(* Logix 5000 project; controller cal1632 1756-L62 rev 16.20; software revision 16.05; part 41 of 61 *)
(* tags used below, declared in another part *)
   FAULT : BOOL;
   p01r09_pb_global_reset : BOOL;
   p02_dint_to_hmi : hmi_dint;
   p24_di_edge_guide_auto : BOOL;
   p24_di_edge_guide_center : BOOL;
   p24_di_edge_guide_left : BOOL;
   p24_di_edge_guide_right : BOOL;
   p24_dint_to_hmi : DINT[16];
   p24_do_edge_guide_input_1 : BOOL;
   p24r01 : routine;
   p24r02 : routine;
   p24r02_fault_exists : BOOL;
   p24r02_timer_fault : TIMER[4];
   p24r02_timer_warning : TIMER[4];
   p24r02_unack_fault : BOOL;
   p24r02_unack_warning : BOOL;
   p24r02_warning_exists : BOOL;
   p24r03 : routine;
   p24r03_timer_fault : TIMER[4];
   p24r03_timer_warning : TIMER[4];
   p24r04 : routine;
   p24r04_timer_fault : TIMER[4];
   p24r04_timer_warning : TIMER[4];
   p24r05 : routine;
   p24r05_timer_fault : TIMER[4];
   p24r05_timer_warning : TIMER[4];
   p24r06 : routine;
   p24r06_timer_fault : TIMER[4];
   p24r06_timer_warning : TIMER[4];
   p24r07 : routine;
   p24r07_timer_fault : TIMER[4];
   p24r07_timer_warning : TIMER[4];
   p24r08 : routine;
   p24r09 : routine;
   p24r10 : routine;

PROGRAM P24_Edge_Control   (* main routine R01_Main *)

ROUTINE R01_Main   (* ladder *)
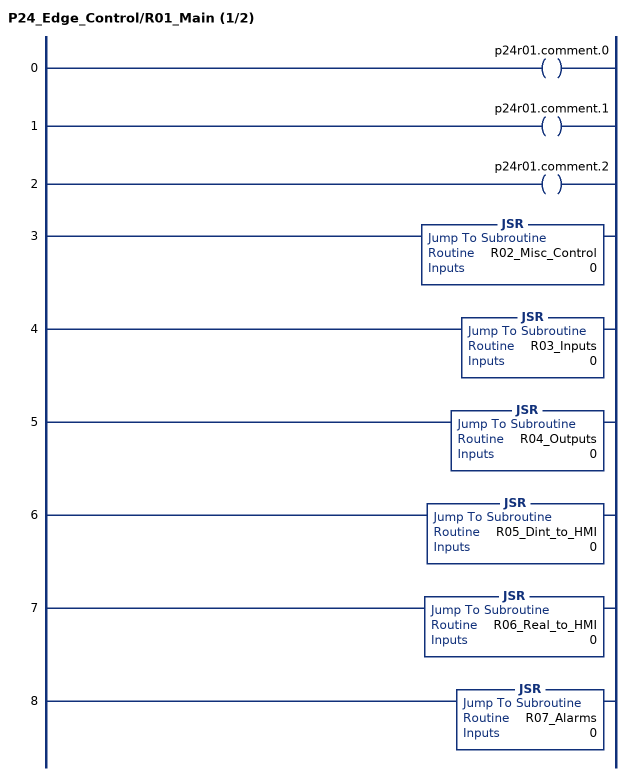
   0: OTE(p24r01.comment.0);
   1: OTE(p24r01.comment.1);
   2: OTE(p24r01.comment.2);
   3: JSR(R02_Misc_Control,0);
   4: JSR(R03_Inputs,0);
   5: JSR(R04_Outputs,0);
   6: JSR(R05_Dint_to_HMI,0);
   7: JSR(R06_Real_to_HMI,0);
   8: JSR(R07_Alarms,0);
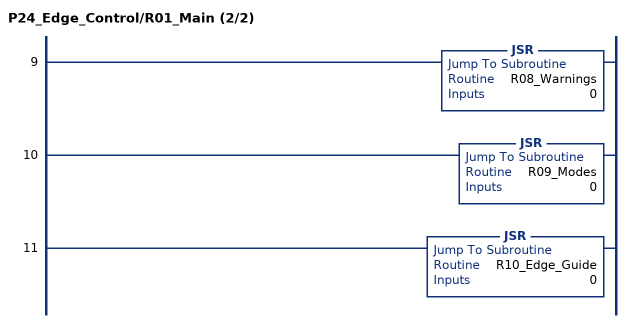
   9: JSR(R08_Warnings,0);
   10: JSR(R09_Modes,0);
   11: JSR(R10_Edge_Guide,0);
END_ROUTINE

ROUTINE R02_Misc_Control   (* ladder *)
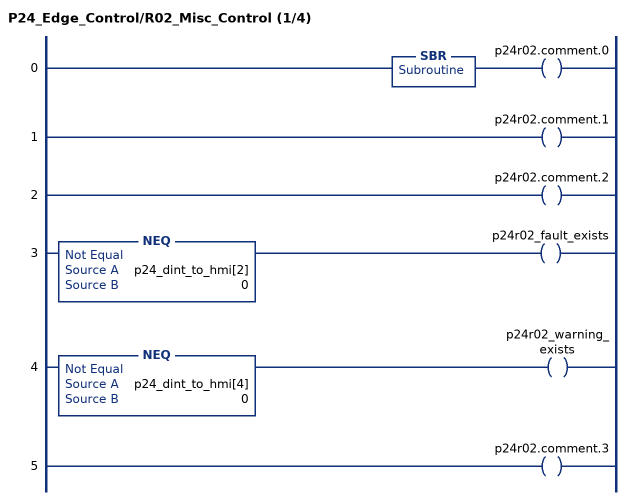
   0: SBR()OTE(p24r02.comment.0);
   1: OTE(p24r02.comment.1);
   2: OTE(p24r02.comment.2);
   3: NEQ(p24_dint_to_hmi[2],0)OTE(p24r02_fault_exists);
   4: NEQ(p24_dint_to_hmi[4],0)OTE(p24r02_warning_exists);
   5: OTE(p24r02.comment.3);
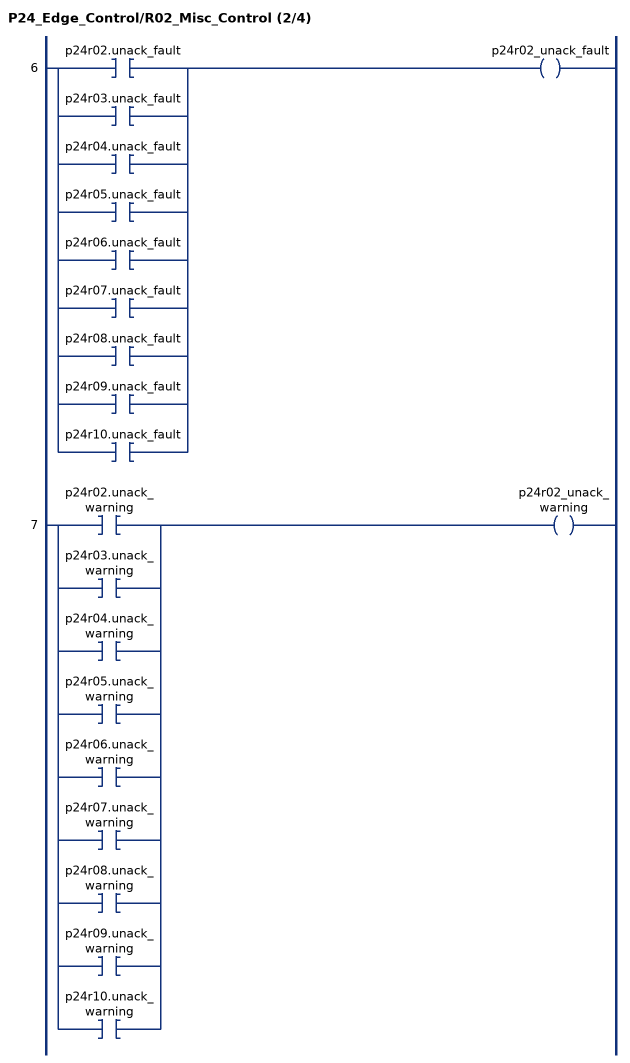
   6: [XIC(p24r02.unack_fault) ,XIC(p24r03.unack_fault) ,XIC(p24r04.unack_fault) ,XIC(p24r05.unack_fault) ,XIC(p24r06.unack_fault) ,XIC(p24r07.unack_fault) ,XIC(p24r08.unack_fault) ,XIC(p24r09.unack_fault) ,XIC(p24r10.unack_fault) ]OTE(p24r02_unack_fault);
   7: [XIC(p24r02.unack_warning) ,XIC(p24r03.unack_warning) ,XIC(p24r04.unack_warning) ,XIC(p24r05.unack_warning) ,XIC(p24r06.unack_warning) ,XIC(p24r07.unack_warning) ,XIC(p24r08.unack_warning) ,XIC(p24r09.unack_warning) ,XIC(p24r10.unack_warning) ]OTE(p24r02_unack_warning);
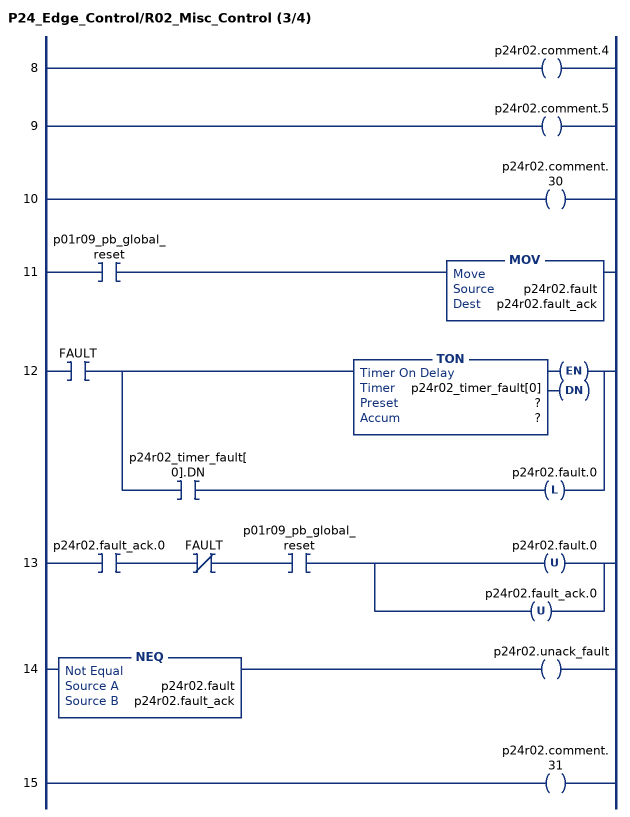
   8: OTE(p24r02.comment.4);
   9: OTE(p24r02.comment.5);
   10: OTE(p24r02.comment.30);
   11: XIC(p01r09_pb_global_reset)MOV(p24r02.fault,p24r02.fault_ack);
   12: XIC(FAULT)[TON(p24r02_timer_fault[0],?,?) ,XIC(p24r02_timer_fault[0].DN) OTL(p24r02.fault.0) ];
   13: XIC(p24r02.fault_ack.0)XIO(FAULT)XIC(p01r09_pb_global_reset)[OTU(p24r02.fault.0) ,OTU(p24r02.fault_ack.0) ];
   14: NEQ(p24r02.fault,p24r02.fault_ack)OTE(p24r02.unack_fault);
   15: OTE(p24r02.comment.31);
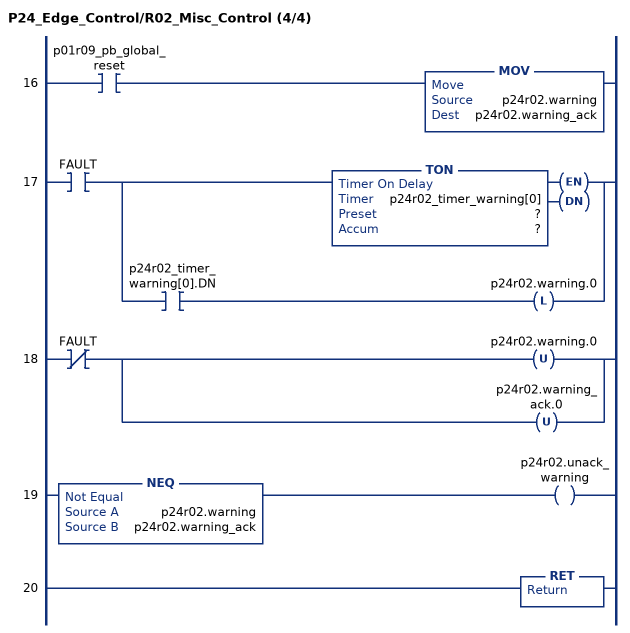
   16: XIC(p01r09_pb_global_reset)MOV(p24r02.warning,p24r02.warning_ack);
   17: XIC(FAULT)[TON(p24r02_timer_warning[0],?,?) ,XIC(p24r02_timer_warning[0].DN) OTL(p24r02.warning.0) ];
   18: XIO(FAULT)[OTU(p24r02.warning.0) ,OTU(p24r02.warning_ack.0) ];
   19: NEQ(p24r02.warning,p24r02.warning_ack)OTE(p24r02.unack_warning);
   20: RET();
END_ROUTINE

ROUTINE R03_Inputs   (* ladder *)
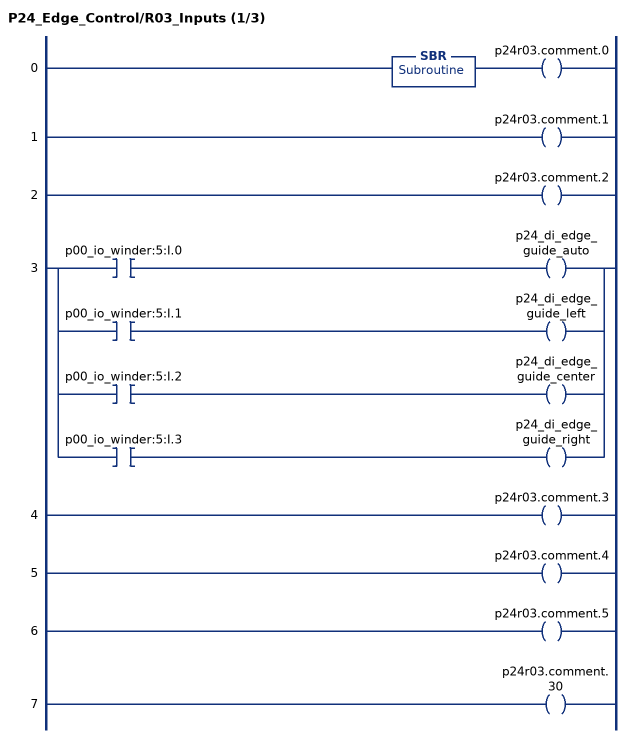
   0: SBR()OTE(p24r03.comment.0);
   1: OTE(p24r03.comment.1);
   2: OTE(p24r03.comment.2);
   3: [XIC(p00_io_winder:5:I.0) OTE(p24_di_edge_guide_auto) ,XIC(p00_io_winder:5:I.1) OTE(p24_di_edge_guide_left) ,XIC(p00_io_winder:5:I.2) OTE(p24_di_edge_guide_center) ,XIC(p00_io_winder:5:I.3) OTE(p24_di_edge_guide_right) ];
   4: OTE(p24r03.comment.3);
   5: OTE(p24r03.comment.4);
   6: OTE(p24r03.comment.5);
   7: OTE(p24r03.comment.30);
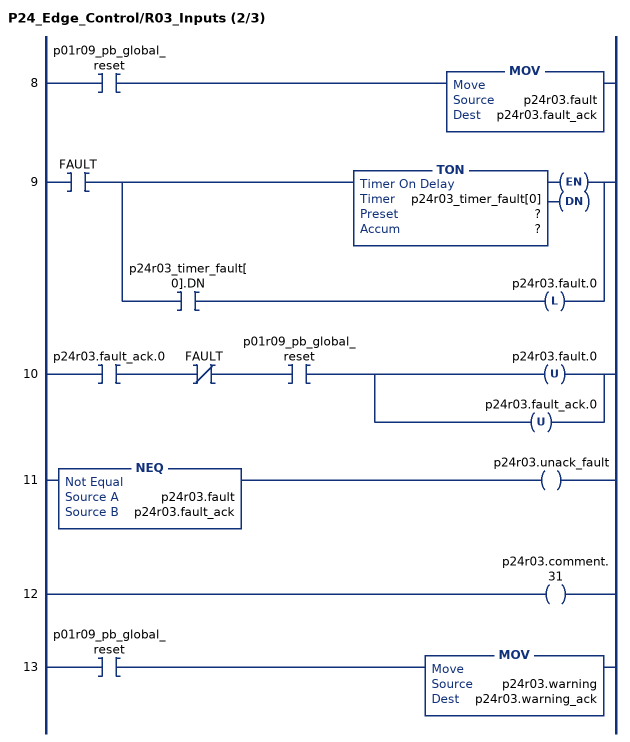
   8: XIC(p01r09_pb_global_reset)MOV(p24r03.fault,p24r03.fault_ack);
   9: XIC(FAULT)[TON(p24r03_timer_fault[0],?,?) ,XIC(p24r03_timer_fault[0].DN) OTL(p24r03.fault.0) ];
   10: XIC(p24r03.fault_ack.0)XIO(FAULT)XIC(p01r09_pb_global_reset)[OTU(p24r03.fault.0) ,OTU(p24r03.fault_ack.0) ];
   11: NEQ(p24r03.fault,p24r03.fault_ack)OTE(p24r03.unack_fault);
   12: OTE(p24r03.comment.31);
   13: XIC(p01r09_pb_global_reset)MOV(p24r03.warning,p24r03.warning_ack);
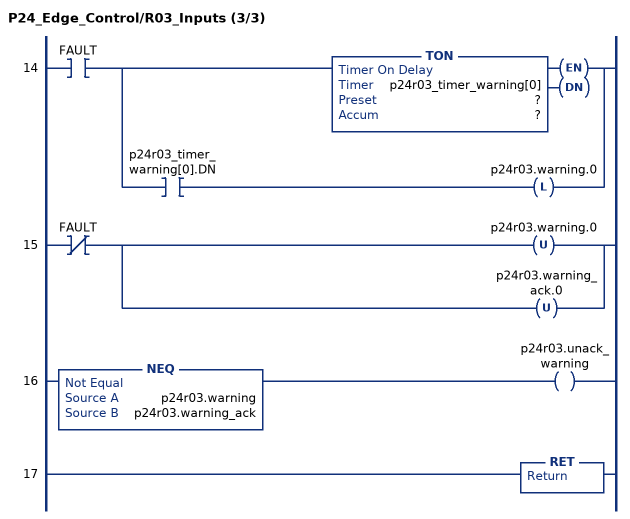
   14: XIC(FAULT)[TON(p24r03_timer_warning[0],?,?) ,XIC(p24r03_timer_warning[0].DN) OTL(p24r03.warning.0) ];
   15: XIO(FAULT)[OTU(p24r03.warning.0) ,OTU(p24r03.warning_ack.0) ];
   16: NEQ(p24r03.warning,p24r03.warning_ack)OTE(p24r03.unack_warning);
   17: RET();
END_ROUTINE

ROUTINE R04_Outputs   (* ladder *)
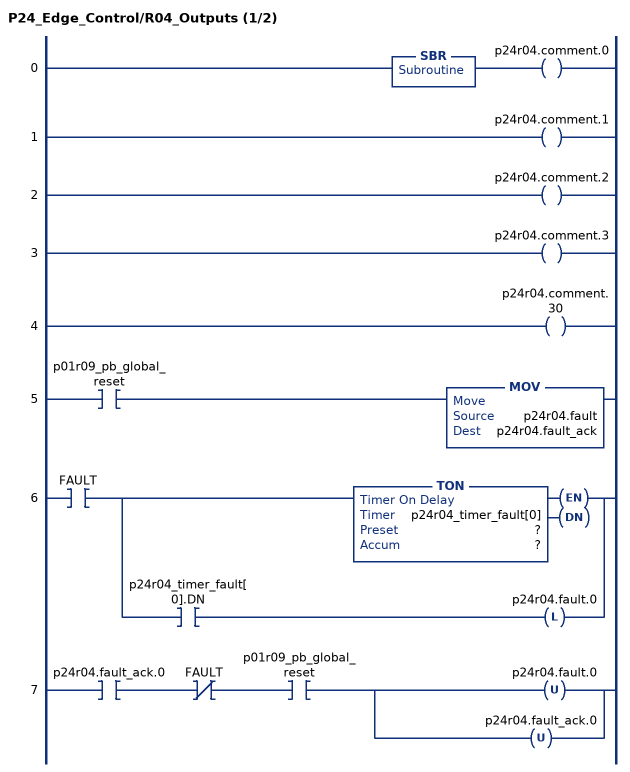
   0: SBR()OTE(p24r04.comment.0);
   1: OTE(p24r04.comment.1);
   2: OTE(p24r04.comment.2);
   3: OTE(p24r04.comment.3);
   4: OTE(p24r04.comment.30);
   5: XIC(p01r09_pb_global_reset)MOV(p24r04.fault,p24r04.fault_ack);
   6: XIC(FAULT)[TON(p24r04_timer_fault[0],?,?) ,XIC(p24r04_timer_fault[0].DN) OTL(p24r04.fault.0) ];
   7: XIC(p24r04.fault_ack.0)XIO(FAULT)XIC(p01r09_pb_global_reset)[OTU(p24r04.fault.0) ,OTU(p24r04.fault_ack.0) ];
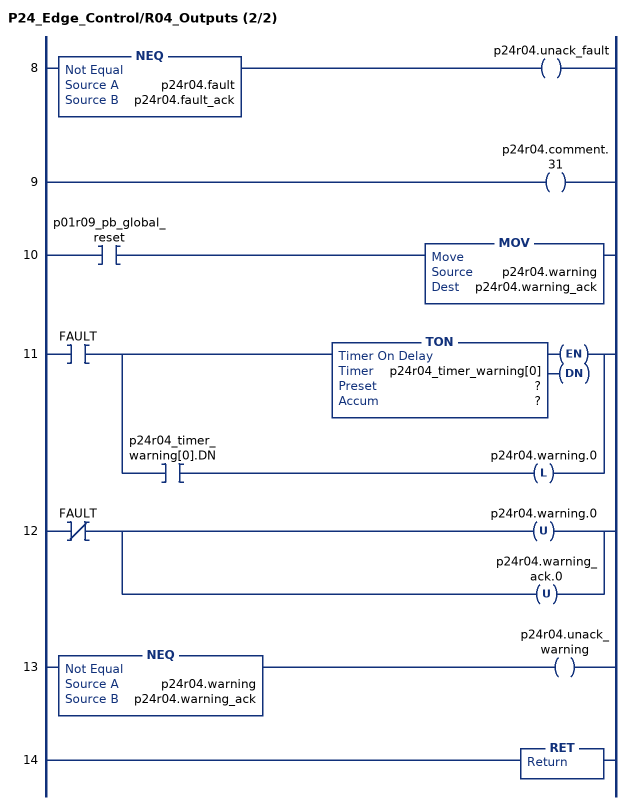
   8: NEQ(p24r04.fault,p24r04.fault_ack)OTE(p24r04.unack_fault);
   9: OTE(p24r04.comment.31);
   10: XIC(p01r09_pb_global_reset)MOV(p24r04.warning,p24r04.warning_ack);
   11: XIC(FAULT)[TON(p24r04_timer_warning[0],?,?) ,XIC(p24r04_timer_warning[0].DN) OTL(p24r04.warning.0) ];
   12: XIO(FAULT)[OTU(p24r04.warning.0) ,OTU(p24r04.warning_ack.0) ];
   13: NEQ(p24r04.warning,p24r04.warning_ack)OTE(p24r04.unack_warning);
   14: RET();
END_ROUTINE

ROUTINE R05_Dint_to_HMI   (* ladder *)
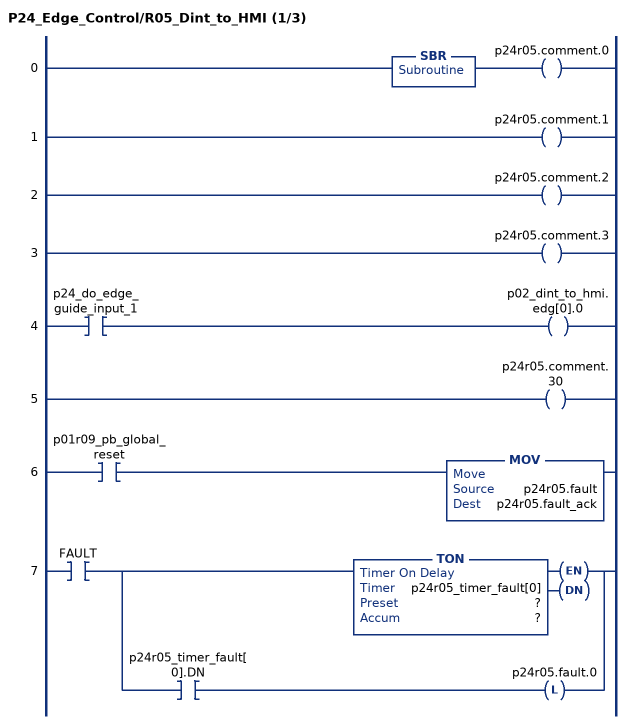
   0: SBR()OTE(p24r05.comment.0);
   1: OTE(p24r05.comment.1);
   2: OTE(p24r05.comment.2);
   3: OTE(p24r05.comment.3);
   4: XIC(p24_do_edge_guide_input_1)OTE(p02_dint_to_hmi.edg[0].0);
   5: OTE(p24r05.comment.30);
   6: XIC(p01r09_pb_global_reset)MOV(p24r05.fault,p24r05.fault_ack);
   7: XIC(FAULT)[TON(p24r05_timer_fault[0],?,?) ,XIC(p24r05_timer_fault[0].DN) OTL(p24r05.fault.0) ];
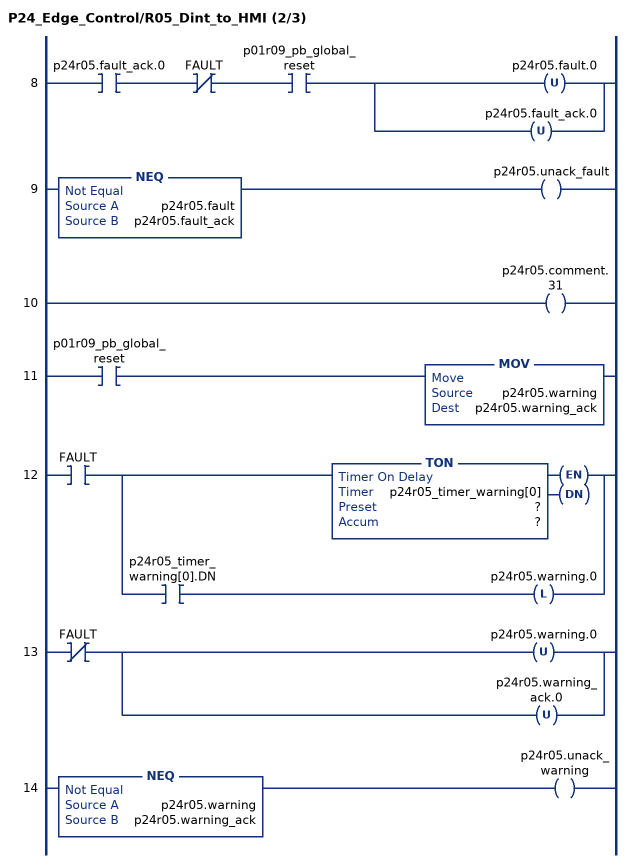
   8: XIC(p24r05.fault_ack.0)XIO(FAULT)XIC(p01r09_pb_global_reset)[OTU(p24r05.fault.0) ,OTU(p24r05.fault_ack.0) ];
   9: NEQ(p24r05.fault,p24r05.fault_ack)OTE(p24r05.unack_fault);
   10: OTE(p24r05.comment.31);
   11: XIC(p01r09_pb_global_reset)MOV(p24r05.warning,p24r05.warning_ack);
   12: XIC(FAULT)[TON(p24r05_timer_warning[0],?,?) ,XIC(p24r05_timer_warning[0].DN) OTL(p24r05.warning.0) ];
   13: XIO(FAULT)[OTU(p24r05.warning.0) ,OTU(p24r05.warning_ack.0) ];
   14: NEQ(p24r05.warning,p24r05.warning_ack)OTE(p24r05.unack_warning);
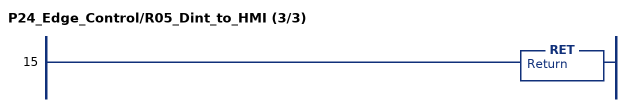
   15: RET();
END_ROUTINE

ROUTINE R06_Real_to_HMI   (* ladder *)
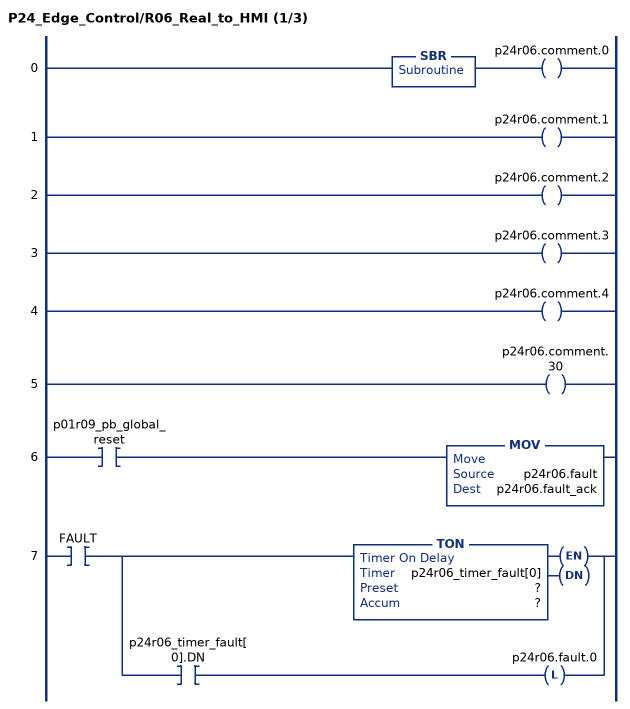
   0: SBR()OTE(p24r06.comment.0);
   1: OTE(p24r06.comment.1);
   2: OTE(p24r06.comment.2);
   3: OTE(p24r06.comment.3);
   4: OTE(p24r06.comment.4);
   5: OTE(p24r06.comment.30);
   6: XIC(p01r09_pb_global_reset)MOV(p24r06.fault,p24r06.fault_ack);
   7: XIC(FAULT)[TON(p24r06_timer_fault[0],?,?) ,XIC(p24r06_timer_fault[0].DN) OTL(p24r06.fault.0) ];
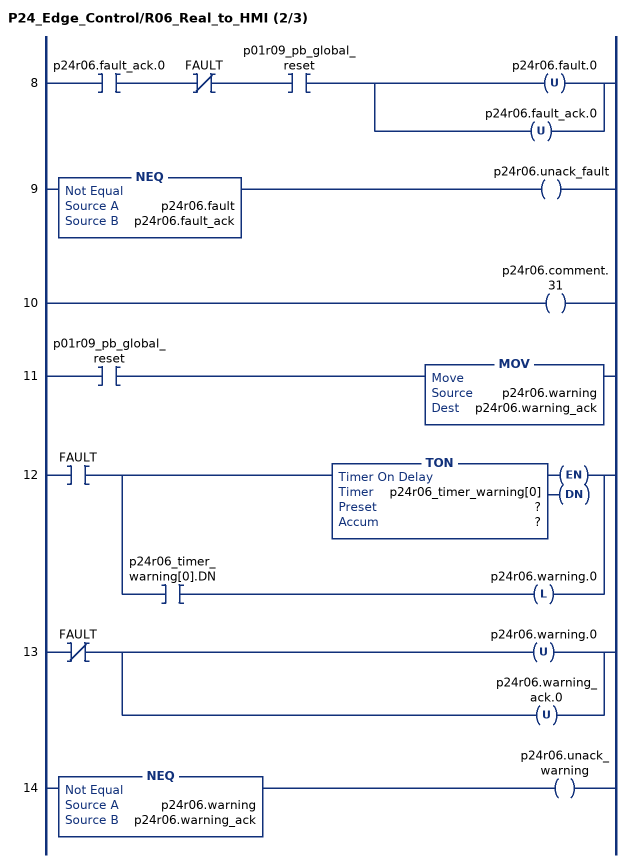
   8: XIC(p24r06.fault_ack.0)XIO(FAULT)XIC(p01r09_pb_global_reset)[OTU(p24r06.fault.0) ,OTU(p24r06.fault_ack.0) ];
   9: NEQ(p24r06.fault,p24r06.fault_ack)OTE(p24r06.unack_fault);
   10: OTE(p24r06.comment.31);
   11: XIC(p01r09_pb_global_reset)MOV(p24r06.warning,p24r06.warning_ack);
   12: XIC(FAULT)[TON(p24r06_timer_warning[0],?,?) ,XIC(p24r06_timer_warning[0].DN) OTL(p24r06.warning.0) ];
   13: XIO(FAULT)[OTU(p24r06.warning.0) ,OTU(p24r06.warning_ack.0) ];
   14: NEQ(p24r06.warning,p24r06.warning_ack)OTE(p24r06.unack_warning);
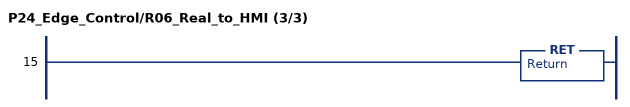
   15: RET();
END_ROUTINE

ROUTINE R07_Alarms   (* ladder *)
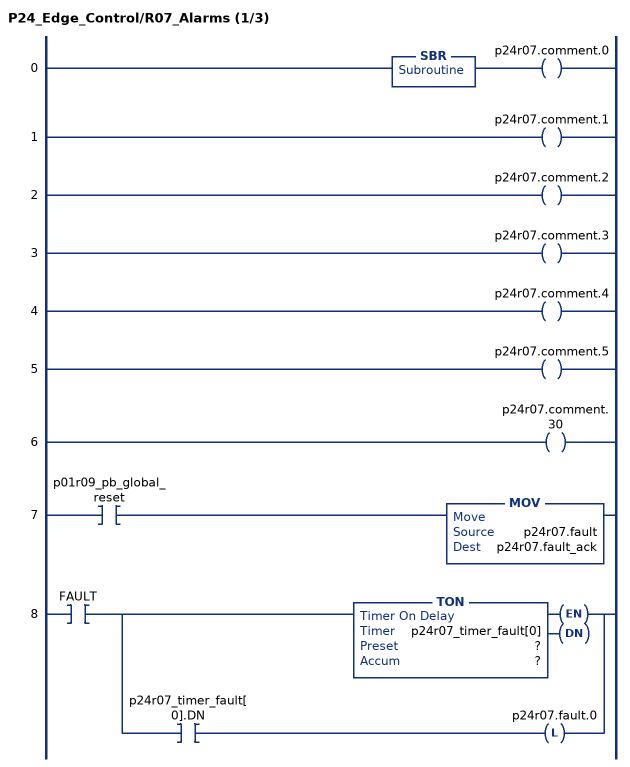
   0: SBR()OTE(p24r07.comment.0);
   1: OTE(p24r07.comment.1);
   2: OTE(p24r07.comment.2);
   3: OTE(p24r07.comment.3);
   4: OTE(p24r07.comment.4);
   5: OTE(p24r07.comment.5);
   6: OTE(p24r07.comment.30);
   7: XIC(p01r09_pb_global_reset)MOV(p24r07.fault,p24r07.fault_ack);
   8: XIC(FAULT)[TON(p24r07_timer_fault[0],?,?) ,XIC(p24r07_timer_fault[0].DN) OTL(p24r07.fault.0) ];
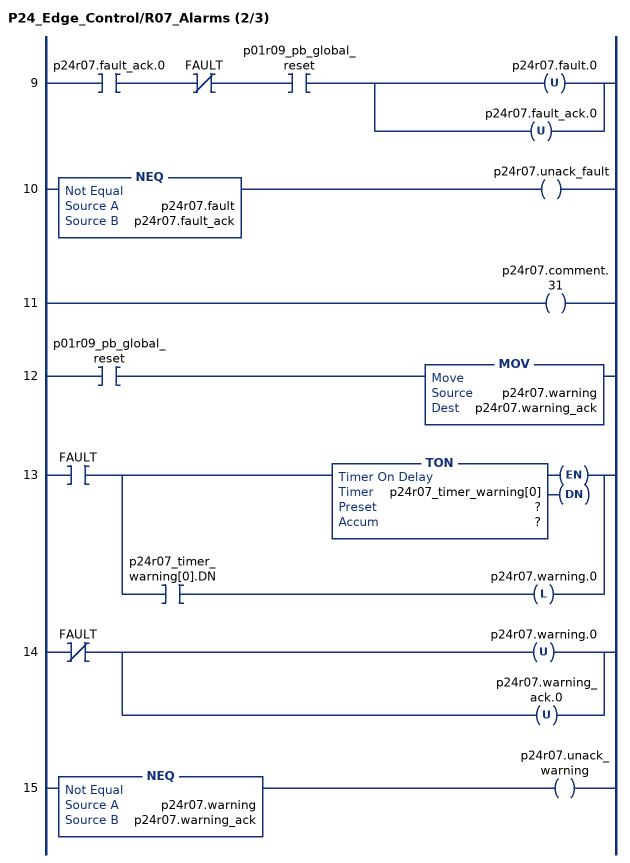
   9: XIC(p24r07.fault_ack.0)XIO(FAULT)XIC(p01r09_pb_global_reset)[OTU(p24r07.fault.0) ,OTU(p24r07.fault_ack.0) ];
   10: NEQ(p24r07.fault,p24r07.fault_ack)OTE(p24r07.unack_fault);
   11: OTE(p24r07.comment.31);
   12: XIC(p01r09_pb_global_reset)MOV(p24r07.warning,p24r07.warning_ack);
   13: XIC(FAULT)[TON(p24r07_timer_warning[0],?,?) ,XIC(p24r07_timer_warning[0].DN) OTL(p24r07.warning.0) ];
   14: XIO(FAULT)[OTU(p24r07.warning.0) ,OTU(p24r07.warning_ack.0) ];
   15: NEQ(p24r07.warning,p24r07.warning_ack)OTE(p24r07.unack_warning);
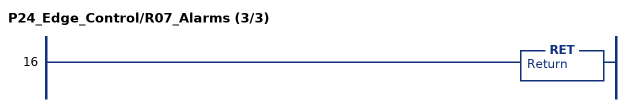
   16: RET();
END_ROUTINE
